FUNCTION_BLOCK MUL_LINT (* IEC 61131-3 LINT Multiplication *)
  (* Standard: 61131-3 *)
  (* Version 0.0, 2004-12-15, JHC, Rockwell Automation, Converted from SRC format. *)
  (* Compiler header: package fb.rt.plc.math; *)
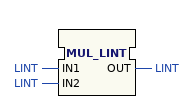
  VAR_INPUT
    IN1 : LINT; (* Multiplicand *)
    IN2 : LINT; (* Multiplier *)
  END_VAR
  VAR_OUTPUT
    OUT : LINT; (* Product *)
  END_VAR
END_FUNCTION_BLOCK
